(* PLC project BasicCoR_PLC, Beckhoff Automation GmbH TwinCAT PLC Control 3.5.13.21 *)
(* stored: creationDateTime 2024-01-02T12:18:06.6022499, modificationDateTime 2024-01-02T12:18:06.6084642 *)

INTERFACE I_Handler
METHOD handle : BOOL
VAR_INPUT
	request	:	STRING;
END_VAR
END_METHOD
METHOD setNext : BOOL
VAR_INPUT
	h	: I_Handler;
END_VAR
END_METHOD
END_INTERFACE

FUNCTION_BLOCK FB_BaseHandler IMPLEMENTS I_Handler
VAR_INPUT
END_VAR
VAR_OUTPUT
END_VAR
VAR
	next : I_Handler;
END_VAR

                  
                

METHOD handle : BOOL
VAR_INPUT
	request	:	STRING;
END_VAR
                        IF ADR(next) <> 0 THEN
	next.handle(request);
END_IF
                      
END_METHOD

METHOD setNext : BOOL
VAR_INPUT
	h	: I_Handler;
END_VAR
                        next := h;
                      
END_METHOD
END_FUNCTION_BLOCK

FUNCTION_BLOCK FB_StaticHandler1 EXTENDS FB_BaseHandler
VAR_INPUT
END_VAR
VAR_OUTPUT
END_VAR
VAR
END_VAR

                  
                

METHOD handle : BOOL
VAR_INPUT
	request	:	STRING;
END_VAR
                        IF request = 'Handler 1 Interupt' THEN
	ADSLOGSTR(ADSLOG_MSGTYPE_MSGBOX, request, ' ');
ELSE
	ADSLOGSTR(ADSLOG_MSGTYPE_MSGBOX, '@H1 Moving to next handler ', '');
	SUPER^.handle(request);
END_IF
                      
END_METHOD
END_FUNCTION_BLOCK

FUNCTION_BLOCK FB_StaticHandler2 EXTENDS FB_BaseHandler
VAR_INPUT
END_VAR
VAR_OUTPUT
END_VAR
VAR
END_VAR

                  
                

METHOD handle : BOOL
VAR_INPUT
	request	:	STRING;
END_VAR
                        IF request = 'Handler 2 Interupt' THEN
	ADSLOGSTR(ADSLOG_MSGTYPE_MSGBOX, request, ' ');
ELSE
	ADSLOGSTR(ADSLOG_MSGTYPE_MSGBOX, '@H2 Moving to next handler ', '');
	SUPER^.handle(request);
END_IF
                      
END_METHOD
END_FUNCTION_BLOCK

FUNCTION_BLOCK FB_StaticHandler3 EXTENDS FB_BaseHandler
VAR_INPUT
END_VAR
VAR_OUTPUT
END_VAR
VAR
END_VAR

                  
                

METHOD handle : BOOL
VAR_INPUT
	request	:	STRING;
END_VAR
                        IF request = 'Handler 3 Interupt' THEN
	ADSLOGSTR(ADSLOG_MSGTYPE_MSGBOX, request, ' ');
ELSE
	ADSLOGSTR(ADSLOG_MSGTYPE_MSGBOX, '@H3 Moving to next handler ', '');
	SUPER^.handle(request);
END_IF
                      
END_METHOD
END_FUNCTION_BLOCK

FUNCTION_BLOCK FB_StaticHandler_n EXTENDS FB_BaseHandler
VAR_INPUT
END_VAR
VAR_OUTPUT
END_VAR
VAR
END_VAR

                  
                

METHOD handle : BOOL
VAR_INPUT
	request	:	STRING;
END_VAR
                        ADSLOGSTR(ADSLOG_MSGTYPE_MSGBOX, request , '');

                      
END_METHOD
END_FUNCTION_BLOCK

PROGRAM MAIN
VAR
	h1				:	FB_StaticHandler1;
	h2				:	FB_StaticHandler2;
	h3				:	FB_StaticHandler3;
	h_n				:	FB_StaticHandler_n;
	request 		:	STRING	:= 'Hello world!';
	xStartProcess	: 	BOOL;
END_VAR

                  h1.setNext(h2);
h2.setNext(h3);
h3.setNext(h_n);

(*************************************************************
*************SIMULATION***************************************
***
*** Leave request as "hello world!" for full chain processing
*** or use the string phrases below to interupt the chain.
***
***	Handler 1 - request := 'Handler 1 Interupt';
*** Handler 2 - request := 'Handler 2 Interupt';
*** Handler 3 - request := 'Handler 3 Interupt';
**************************************************************
*************************************************************)

IF xStartProcess THEN
	xStartProcess := FALSE;
	h1.handle(request);
END_IF

                
END_PROGRAM

CONFIGURATION Application
  RESOURCE BasicCoR_PLC ON PLC
    TASK PlcTask(INTERVAL := T#0ms, PRIORITY := 20);
    PROGRAM MAIN WITH PlcTask : MAIN;
  END_RESOURCE
END_CONFIGURATION
